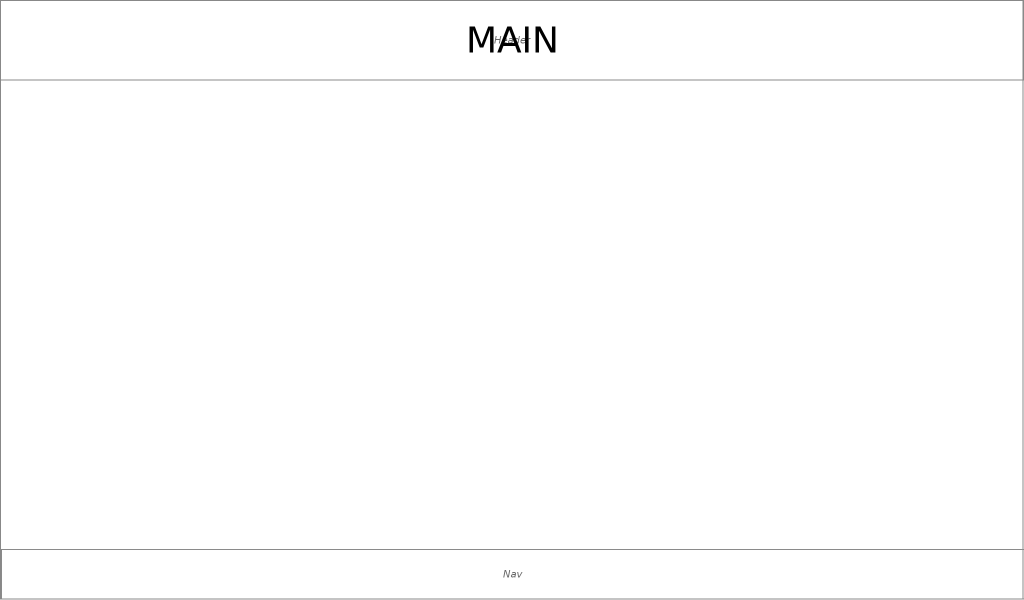
VISUALIZATION MainScreen  // 1024x600
    Frame (0,0 1024x80)
        shows Header()
    Frame (1,549 1024x50)
        shows Nav()
    Label (334,16 357x48), "MAIN"
END_VISUALIZATION

(* stored: Version 1.1.0.1, ProductVersion 3.1.4024.12
   Visu MainScreen: Id {ded18176-b6f4-4194-a37d-67b79222977a} *)
